Yaskawa INFORM job: SkinDetect.JBI

/JOB
//NAME SkinDetect
//POS
///NPOS 7,0,0,0,0,0
///TOOL 0
///POSTYPE PULSE
///PULSE
C00000=-7969,21694,-5134,1465,-52599,3149
C00001=-8763,22537,-40304,2696,-23898,2515
C00002=18727,25090,-37193,-1570,-24960,-7959
C00003=13881,45329,-12162,-664,-32902,-6224
C00004=-6835,42752,-15687,1905,-31515,2123
C00005=-8763,22537,-40304,2696,-23898,2515
C00006=-7969,21694,-5134,1465,-52599,3149
//INST
///DATE 2026/05/05 16:03
///ATTR SC,RW
///GROUP1 RB1
NOP
MOVJ C00000 VJ=0.78
MOVJ C00001 VJ=0.78
MOVL C00002 V=11.0
MOVL C00003 V=11.0
MOVL C00004 V=11.0
MOVL C00005 V=11.0
MOVJ C00006 VJ=0.78
END
